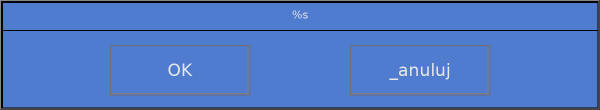
VISUALIZATION D_DeleteRecipeCleim  // 600x110
VAR_IN_OUT
	stData : ST_MCHMIPrepareScreen_02_XX_DeleteRecipe;
END_VAR
    Rectangle (0,0 600x110)
    Line (0,30) (600,30)
    Rectangle (3,3 594x24), "%s", text variable: stData.wsNameRecipe, text list: 'TextList_02', text index: 0
    Button (350,45 140x50), "_anuluj", text list: 'TextListGlobal', text index: 2
        OnMouseDown: execute { stData.bCancel := TRUE; }
        OnMouseUp: CloseDialog Dialog=D_DeleteRecipeCleim, Result=Ignore, NumpadKeypadSet=True
    Button (110,45 140x50), "OK"
        OnMouseDown: execute { stData.bOK := TRUE; }
        OnMouseUp: CloseDialog Dialog=D_DeleteRecipeCleim, Result=OK, NumpadKeypadSet=True
END_VISUALIZATION

(* stored: Version 1.1.0.1
   Visu D_DeleteRecipeCleim: Id {522b2c91-7cfd-0101-3310-cc0831e46d8a} *)
